// TIA Portal V15.1 export
// export: Created 2024-06-21T08:41:03.3487684Z, ExportSetting WithDefaults, DisplayName Totally Integrated Automation Portal, DisplayVersion V15.1 Update 5, DisplayName TIA Portal Openness, DisplayVersion V15.1 Update 5, DisplayName SINAMICS Startdrive Advanced, DisplayVersion V15.1, DisplayName G130, G150, S120, S150, SINAMICS MV, S210, DisplayVersion V15.1, DisplayName G110M, G120, G120C, G120D, G120P, DisplayVersion V15.1, DisplayName STEP 7 Professional, DisplayVersion V15.1 Update 5, DisplayName STEP 7 Safety, DisplayVersion V15.1, DisplayName WinCC Professional, DisplayVersion V15.1 Update 5, DisplayName SIMATIC Visualization Architect, DisplayVersion V15.1
FUNCTION_BLOCK "LProcMot1W-FCByp"   // FB1728, FBD
TITLE = LProcMotFCPidNoFbk
{ S7_Optimized_Access := 'FALSE' }
AUTHOR : VCC
FAMILY : ProcEq
NAME : FCPN
VERSION : 0.0
// ===============================================================================
// 
// This "Motor-1Way-1Speed-FreqCtrl with bypass module is used in applications 
// when 
// a motor 
// 1 way - 1 speed equipped with Danfoss equipment (FC) on
// Profibus or Profinet steering is needed.
// The module contains: 
// " 1selection 5 set point with 5 resonance 
// "1 mode from HMI
// "1 motor protection.
// "1 safety switch.
// "1 feedback motor running (option): Pressure-switch, Rotation guard,........
// "1 Proces Danfoss equipment with Profibus/Profinet.
// "1 bypass contactor.
// "1 bypass key-switch.
// ===============================================================================
// stored: AutoNumber false, IsIECCheckEnabled false, SetENOAutomatically False, UDAEnableTagReadback false
   VAR_INPUT
      I_ExtSP1_Value { ExternalAccessible := 'False'; ExternalVisible := 'False'; ExternalWritable := 'False'} : Real;   // External Set-point 1
      I_SPReq : Int;   // Index Set-point Request
      I_ExtSP1 { ExternalAccessible := 'False'; ExternalVisible := 'False'; ExternalWritable := 'False'} : Bool;   // External Set-point 1 Request
      I_EnableFCReset { ExternalAccessible := 'False'; ExternalVisible := 'False'; ExternalWritable := 'False'} : Bool;   // Enable Frequency reset with Fielbus
      I_EnableCheckSpeedOK { ExternalAccessible := 'False'; ExternalVisible := 'False'; ExternalWritable := 'False'} : Bool;   // Enable check speed is OK
      I_TimeCheckSpeedOK { ExternalAccessible := 'False'; ExternalVisible := 'False'; ExternalWritable := 'False'} : DInt := DINT#10000;   // Delay time to check if speed is OK
      I_RunFbkAlarmTime { ExternalAccessible := 'False'; ExternalVisible := 'False'; ExternalWritable := 'False'} : DInt;   // Time for alarm Feedback Motor running
      I_EnableAlarm { ExternalAccessible := 'False'; ExternalVisible := 'False'; ExternalWritable := 'False'} : Bool;   // Enable alarm
      I_AutoReq { ExternalAccessible := 'False'; ExternalVisible := 'False'; ExternalWritable := 'False'} : Bool;   // Auto Request from equation or Sequence
      I_InterlockOk { ExternalAccessible := 'False'; ExternalVisible := 'False'; ExternalWritable := 'False'} : Bool;   // Interlock Ok
      I_MotorProtection { ExternalAccessible := 'False'; ExternalVisible := 'False'; ExternalWritable := 'False'} : Bool;   // Motor protection Ok
      I_BypassKey { ExternalAccessible := 'False'; ExternalVisible := 'False'; ExternalWritable := 'False'} : Bool;   // Bypass Key-switch
      I_SafetySwitch { ExternalAccessible := 'False'; ExternalVisible := 'False'; ExternalWritable := 'False'} : Bool;   // Safety Switch Ok
      I_RunFeedBack { ExternalAccessible := 'False'; ExternalVisible := 'False'; ExternalWritable := 'False'} : Bool;   // Feedback motor running (Pressure-switch, Rotation Guard,...)
      I_PBSetPBResetAllAutoSel { ExternalAccessible := 'False'; ExternalVisible := 'False'; ExternalWritable := 'False'} : Struct   // Set PB activated - Reset PB activated - All HMI Auto selected
         HMI1SetPB { ExternalAccessible := 'False'; ExternalVisible := 'False'; ExternalWritable := 'False'} : Bool;   // Set PB activated on HMI1
         HMI1ResetPB { ExternalAccessible := 'False'; ExternalVisible := 'False'; ExternalWritable := 'False'} : Bool;   // Reset PB activated on HMI1
         HMI1AllHMIAutoSel { ExternalAccessible := 'False'; ExternalVisible := 'False'; ExternalWritable := 'False'} : Bool;   // All HMI Auto selected on HMI1
         HMI2SetPB { ExternalAccessible := 'False'; ExternalVisible := 'False'; ExternalWritable := 'False'} : Bool;   // Set PB activated on HMI2
         HMI2ResetPB { ExternalAccessible := 'False'; ExternalVisible := 'False'; ExternalWritable := 'False'} : Bool;   // Reset PB activated on HMI2
         HMI2AllHMIAutoSel { ExternalAccessible := 'False'; ExternalVisible := 'False'; ExternalWritable := 'False'} : Bool;   // All HMI Auto selected on HMI2
         HMI3SetPB { ExternalAccessible := 'False'; ExternalVisible := 'False'; ExternalWritable := 'False'} : Bool;   // Set PB activated on HMI3
         HMI3ResetPB { ExternalAccessible := 'False'; ExternalVisible := 'False'; ExternalWritable := 'False'} : Bool;   // Reset PB activated on HMI3
         HMI3AllHMIAutoSel { ExternalAccessible := 'False'; ExternalVisible := 'False'; ExternalWritable := 'False'} : Bool;   // All HMI Auto selected on HMI3
         HMI4SetPB { ExternalAccessible := 'False'; ExternalVisible := 'False'; ExternalWritable := 'False'} : Bool;   // Set PB activated on HMI4
         HMI4ResetPB { ExternalAccessible := 'False'; ExternalVisible := 'False'; ExternalWritable := 'False'} : Bool;   // Reset PB activated on HMI4
         HMI4AllHMIAutoSel { ExternalAccessible := 'False'; ExternalVisible := 'False'; ExternalWritable := 'False'} : Bool;   // All HMI Auto selected on HMI4
         HMI5SetPB { ExternalAccessible := 'False'; ExternalVisible := 'False'; ExternalWritable := 'False'} : Bool;   // Set PB activated on HMI5
         HMI5ResetPB { ExternalAccessible := 'False'; ExternalVisible := 'False'; ExternalWritable := 'False'} : Bool;   // Reset PB activated on HMI5
         HMI5AllHMIAutoSel { ExternalAccessible := 'False'; ExternalVisible := 'False'; ExternalWritable := 'False'} : Bool;   // All HMI Auto selected on HMI5
         StartPBSel { ExternalAccessible := 'False'; ExternalVisible := 'False'; ExternalWritable := 'False'} : Bool;   // Start is activated
         AlarmResetPBSel { ExternalAccessible := 'False'; ExternalVisible := 'False'; ExternalWritable := 'False'} : Bool;   // Alarm reset is activated
      END_STRUCT;
      I_UpperLevelAlarmA { ExternalAccessible := 'False'; ExternalVisible := 'False'; ExternalWritable := 'False'} : Bool;   // Upper level alarm A
      I_UpperLevelAlarmB { ExternalAccessible := 'False'; ExternalVisible := 'False'; ExternalWritable := 'False'} : Bool;   // Upper level alarm B
      I_HWSubInput { ExternalAccessible := 'False'; ExternalVisible := 'False'; ExternalWritable := 'False'} : HW_SUBMODULE;   // I/O connection hardware
      I_HWSubOutput { ExternalAccessible := 'False'; ExternalVisible := 'False'; ExternalWritable := 'False'} : HW_SUBMODULE;   // I/O connection hardware
      C_EnableSetResetHMI { ExternalAccessible := 'False'; ExternalVisible := 'False'; ExternalWritable := 'False'} : Bool;   // Enable Set-Reset functions from HMI
      C_SelfHolding { ExternalAccessible := 'False'; ExternalVisible := 'False'; ExternalWritable := 'False'} : Bool := TRUE;   // Enable SelfHolding Command
      C_RunFeedBackUsed { ExternalAccessible := 'False'; ExternalVisible := 'False'; ExternalWritable := 'False'} : Bool;   // Feedback motor running is used
      C_SafetySwNc { ExternalAccessible := 'False'; ExternalVisible := 'False'; ExternalWritable := 'False'} : Bool;   // Safety switch Normally closed
      C_MotorProtectionNc { ExternalAccessible := 'False'; ExternalVisible := 'False'; ExternalWritable := 'False'} : Bool;   // Motor protection Normally closed
      C_BypassSw_HW { ExternalAccessible := 'False'; ExternalVisible := 'False'; ExternalWritable := 'False'} : Bool := TRUE;   // Bypass-switch Hardware (=true) otherwise Software
      C_BypassSwOffFault { ExternalAccessible := 'False'; ExternalVisible := 'False'; ExternalWritable := 'False'} : Bool := TRUE;   // Bypass Switch active when input = False
      C_ManualForced { ExternalAccessible := 'False'; ExternalVisible := 'False'; ExternalWritable := 'False'} : Bool;   // Manual Forced is used (=true)
   END_VAR
   VAR_OUTPUT
      O_SP : Real;   // Setpoint used in controller
      O_Contactor { ExternalAccessible := 'False'; ExternalVisible := 'False'; ExternalWritable := 'False'} : Bool;   // Contactor of motor loop
      O_MotorRunning { ExternalAccessible := 'False'; ExternalVisible := 'False'; ExternalWritable := 'False'} : Bool;   // Motor is running
      O_AlarmABCondition { ExternalAccessible := 'False'; ExternalVisible := 'False'; ExternalWritable := 'False'} : Bool;   // Alarms resetable
      O_AlarmA { ExternalAccessible := 'False'; ExternalVisible := 'False'; ExternalWritable := 'False'} : Bool;   // Alarm A
      O_AlarmB { ExternalAccessible := 'False'; ExternalVisible := 'False'; ExternalWritable := 'False'} : Bool;   // Alarm B
      O_AlarmC { ExternalAccessible := 'False'; ExternalVisible := 'False'; ExternalWritable := 'False'} : Bool;   // Alarm C
      O_AlarmD { ExternalAccessible := 'False'; ExternalVisible := 'False'; ExternalWritable := 'False'} : Bool;   // Alarm D
      H_IAnim { ExternalAccessible := 'False'; ExternalVisible := 'False'; ExternalWritable := 'False'} : Word;   // HMI Animation color of the icon
      H_AlarmWord { ExternalAccessible := 'False'; ExternalVisible := 'False'; ExternalWritable := 'False'} : DWord;   // Alarm Word
   END_VAR
   VAR_IN_OUT
      FCDP : "LProcDanfoss";   // DB of submodule for the Frequency controller
   END_VAR
   VAR DB_SPECIFIC
      AA_MotorProtection { ExternalAccessible := 'False'; ExternalVisible := 'False'; ExternalWritable := 'False'} : Bool;   // Motor Protection alarm
      AA_SafetySwitch { ExternalAccessible := 'False'; ExternalVisible := 'False'; ExternalWritable := 'False'} : Bool;   // Safety Switch alarm
      AA_FreqController { ExternalAccessible := 'False'; ExternalVisible := 'False'; ExternalWritable := 'False'} : Bool;   // Frequency controller alarm A
      AB_RunFeedback { ExternalAccessible := 'False'; ExternalVisible := 'False'; ExternalWritable := 'False'} : Bool;   // Motor Running Feedback Alarm
      AB_OvTimeAutoSel { ExternalAccessible := 'False'; ExternalVisible := 'False'; ExternalWritable := 'False'} : Bool;   // Overtime Auto selected
      AC_FreqController { ExternalAccessible := 'False'; ExternalVisible := 'False'; ExternalWritable := 'False'} : Bool;   // Frequency controller alarm C
      AD_InterlockAlarm { ExternalAccessible := 'False'; ExternalVisible := 'False'; ExternalWritable := 'False'} : Bool;   // Interlock Alarm
      AD_BypassSwitch { ExternalAccessible := 'False'; ExternalVisible := 'False'; ExternalWritable := 'False'} : Bool;   // Bypass-Switch Alarm
      AD_BypassSoftKey { ExternalAccessible := 'False'; ExternalVisible := 'False'; ExternalWritable := 'False'} : Bool;   // Bypass-Key HMI Alarm
      H_HMIModeCmd : Word;   // Mode commands from HMI
      H_ActiveHMI : Int;   // Active HMI
      H_NameActiveHMI : String[25];   // Name of the Active HMI
      H_In : Struct   // HMI
         Normalbandwidthmode : Bool := TRUE;   // Each resonance frequency his own bandwidth
         SPResonance1 : Real;   // Set-point 1 Resonance frequency
         SPResonance2 : Real;   // Set-point 2 Resonance frequency
         SPResonance3 : Real;   // Set-point 3 Resonance frequency
         SPResonance4 : Real;   // Set-point 4 Resonance frequency
         SPBandwidth1 : Real;   // Set-point 1 Bandwidth (for resonance frequency)
         SPBandwidth2 : Real;   // Set-point 2 Bandwidth (for resonance frequency)
         SPBandwidth3 : Real;   // Set-point 3 Bandwidth (for resonance frequency)
         SPBandwidth4 : Real;   // Set-point 4 Bandwidth (for resonance frequency)
      END_STRUCT;
      H_Out : Struct   // HMI
         MotorProtectIAnim : Word;   // HMI Animation color of object
         SafetySwitchIAnim : Word;   // HMI Animation color of object
         FCIAnim : Word;   // HMI Animation color of object
         ContactorIAnim : Word;   // HMI Animation color of object
         BypassSwitchIAnim : Word;   // HMI Animation color of object
         RunFbkIAnim : Word;   // HMI Animation color of object
         Anim : Word;   // HMI Animation word
         Anim2 : Word;   // HMI Animation word
         Anim3 : Bool;   // HMI Animation bool
         DBnr : Int;   // HMI Animation DB number
      END_STRUCT;
      H_InOut : Struct   // HMI
         SetpntAllowed : Bool := TRUE;   // Setpoint is OK and allowed
         Manual_Value : Real;   // Position Setpoint in Manual
         SP1 : Real;   // Set-point 1
         SP2 : Real;   // Set-point 2
         SP3 : Real;   // Set-point 3
         SP4 : Real;   // Set-point 4
         SP5 : Real;   // Set-point 5
      END_STRUCT;
      AutoMode { ExternalAccessible := 'False'; ExternalVisible := 'False'; ExternalWritable := 'False'} : Bool;   // Auto mode
      ManualMode { ExternalAccessible := 'False'; ExternalVisible := 'False'; ExternalWritable := 'False'} : Bool;   // Manual mode
      AutoModeSel { ExternalAccessible := 'False'; ExternalVisible := 'False'; ExternalWritable := 'False'} : Bool;   // Auto Mode Selection from HMI
      ManualModeSel { ExternalAccessible := 'False'; ExternalVisible := 'False'; ExternalWritable := 'False'} : Bool;   // Manual Mode Selection from HMI
      HMISetCmd { ExternalAccessible := 'False'; ExternalVisible := 'False'; ExternalWritable := 'False'} : Bool;   // Set Command on HMI
      HMIResetCmd { ExternalAccessible := 'False'; ExternalVisible := 'False'; ExternalWritable := 'False'} : Bool;   // Reset Command on HMI
      H_FncSelInHMI { ExternalAccessible := 'False'; ExternalVisible := 'False'; ExternalWritable := 'False'} : Bool;   // Manual selection from HMI
      ForcedMan { ExternalAccessible := 'False'; ExternalVisible := 'False'; ExternalWritable := 'False'} : Bool;   // Forced manual active
      OvTimeAutoSel { ExternalAccessible := 'False'; ExternalVisible := 'False'; ExternalWritable := 'False'} : Bool;   // Overtime Auto selected
      OvTimeAutoSelCond { ExternalAccessible := 'False'; ExternalVisible := 'False'; ExternalWritable := 'False'} : Bool;   // Overtime Auto selected condition
      MotorProtectionABCond { ExternalAccessible := 'False'; ExternalVisible := 'False'; ExternalWritable := 'False'} : Bool;   // Motor protection alarm can be reset
      MotorProtectionDisable { ExternalAccessible := 'False'; ExternalVisible := 'False'; ExternalWritable := 'False'} : Bool;   // Motor protection alarm is disabled from HMI
      SafetySwitchABCond { ExternalAccessible := 'False'; ExternalVisible := 'False'; ExternalWritable := 'False'} : Bool;   // Safety Switch alarm can be reset
      SafetySwitchDisable { ExternalAccessible := 'False'; ExternalVisible := 'False'; ExternalWritable := 'False'} : Bool;   // Safety Switch alarm is disabled from HMI
      StartCmdFC { ExternalAccessible := 'False'; ExternalVisible := 'False'; ExternalWritable := 'False'} : Bool;   // Start Command Frequency controller signal
      MRV_FC { ExternalAccessible := 'False'; ExternalVisible := 'False'; ExternalWritable := 'False'} : Int;   // Frequency controller MRV (main reference value)
      FCActive { ExternalAccessible := 'False'; ExternalVisible := 'False'; ExternalWritable := 'False'} : Bool;   // Frequency controller - Profibus active
      FCAlarmDisable { ExternalAccessible := 'False'; ExternalVisible := 'False'; ExternalWritable := 'False'} : Bool;   // Frequency controller alarms are disable from HMI
      FCABCond { ExternalAccessible := 'False'; ExternalVisible := 'False'; ExternalWritable := 'False'} : Bool;   // Frequency controller alarm can be reset
      BypassSwitchDisable { ExternalAccessible := 'False'; ExternalVisible := 'False'; ExternalWritable := 'False'} : Bool;   // Bypass-switch alarm is disabled from HMI
      BypassForced { ExternalAccessible := 'False'; ExternalVisible := 'False'; ExternalWritable := 'False'} : Bool;   // Bypass Forced by Key-switch
      RunFbkEnAlarm { ExternalAccessible := 'False'; ExternalVisible := 'False'; ExternalWritable := 'False'} : Bool;   // Motor Running Feedback Enable Alarm
      RunFbkDisable { ExternalAccessible := 'False'; ExternalVisible := 'False'; ExternalWritable := 'False'} : Bool;   // Motor Running Feedback Alarm is disabled from HMI
      RunFeedBackABCond { ExternalAccessible := 'False'; ExternalVisible := 'False'; ExternalWritable := 'False'} : Bool;   // Motor Running Feedback Alarm can be reset
      CmdRequest { ExternalAccessible := 'False'; ExternalVisible := 'False'; ExternalWritable := 'False'} : Bool;   // Command request to activate the component
      SetPBMan { ExternalAccessible := 'False'; ExternalVisible := 'False'; ExternalWritable := 'False'} : Bool;   // Set pushbutton is activated in manual
      ResetPBMan { ExternalAccessible := 'False'; ExternalVisible := 'False'; ExternalWritable := 'False'} : Bool;   // Reset pushbutton is activated in manual
      AllHMIAutoSel { ExternalAccessible := 'False'; ExternalVisible := 'False'; ExternalWritable := 'False'} : Bool;   // All HMI Auto selected
      Active { ExternalAccessible := 'False'; ExternalVisible := 'False'; ExternalWritable := 'False'} : Bool;   // Motor Loop is active
      Contactor { ExternalAccessible := 'False'; ExternalVisible := 'False'; ExternalWritable := 'False'} : Bool;   // Contactor
      SPSel { ExternalAccessible := 'False'; ExternalVisible := 'False'; ExternalWritable := 'False'} : Real;   // Set-point selected
      SPReal { ExternalAccessible := 'False'; ExternalVisible := 'False'; ExternalWritable := 'False'} : Real;   // Manual or Automatic Set-point selected Real
      SPDINT { ExternalAccessible := 'False'; ExternalVisible := 'False'; ExternalWritable := 'False'} : DInt;   // Set-point selected DInteger
      AlarmA { ExternalAccessible := 'False'; ExternalVisible := 'False'; ExternalWritable := 'False'} : Bool;   // Summation Alarm A
      AlarmB { ExternalAccessible := 'False'; ExternalVisible := 'False'; ExternalWritable := 'False'} : Bool;   // Summation Alarm B
      AlarmC { ExternalAccessible := 'False'; ExternalVisible := 'False'; ExternalWritable := 'False'} : Bool;   // Summation Alarm C
      AlarmD { ExternalAccessible := 'False'; ExternalVisible := 'False'; ExternalWritable := 'False'} : Bool;   // Summation Alarm D
      DBnr { ExternalAccessible := 'False'; ExternalVisible := 'False'; ExternalWritable := 'False'} : Int;   // HMI DB number
   END_VAR
   VAR
      RunFbkTimer { ExternalAccessible := 'False'; ExternalVisible := 'False'; ExternalWritable := 'False'; S7_SetPoint := 'True'} : "LTimer";   // Timer Run Feedback Alarm
      RunFeedback { ExternalAccessible := 'False'; ExternalVisible := 'False'; ExternalWritable := 'False'; S7_SetPoint := 'True'} : "LProc1AlarmMultiIn";   // Run Feedback Alarm
      MotorProtection { ExternalAccessible := 'False'; ExternalVisible := 'False'; ExternalWritable := 'False'; S7_SetPoint := 'True'} : "LProc1AlarmMultiIn";   // Motor protection alarm
      SafetySwitch { ExternalAccessible := 'False'; ExternalVisible := 'False'; ExternalWritable := 'False'; S7_SetPoint := 'True'} : "LProc1AlarmMultiIn";   // Safety Switch alarm
      BypassSwitch { ExternalAccessible := 'False'; ExternalVisible := 'False'; ExternalWritable := 'False'; S7_SetPoint := 'True'} : "LProc1AlarmMultiIn";   // Bypass alarm
      Modes { ExternalAccessible := 'False'; ExternalVisible := 'False'; ExternalWritable := 'False'; S7_SetPoint := 'True'} : "LProcObjectMode";   // Modes Handling
      SelSp { ExternalAccessible := 'False'; ExternalVisible := 'False'; ExternalWritable := 'False'; S7_SetPoint := 'True'} : "LProcSel5SPResFreq";
   END_VAR
   VAR DB_SPECIFIC
      CheckActiveHMI { ExternalAccessible := 'False'; ExternalVisible := 'False'; ExternalWritable := 'False'; S7_SetPoint := 'True'} : TP_TIME;   // Timer
      CheckActiveHMI_1 { ExternalAccessible := 'False'; ExternalVisible := 'False'; ExternalWritable := 'False'; S7_SetPoint := 'True'} : TP_TIME;   // Timer
      CheckActiveHMI_2 { ExternalAccessible := 'False'; ExternalVisible := 'False'; ExternalWritable := 'False'; S7_SetPoint := 'True'} : TON_TIME;   // Timer
      CheckActiveHMI_3 { ExternalAccessible := 'False'; ExternalVisible := 'False'; ExternalWritable := 'False'; S7_SetPoint := 'True'} : TON_TIME;   // Timer
   END_VAR
   VAR_TEMP
      __PlcmigTempFillBits_0B0 : Array[0..23] of Bool;
   END_VAR
BEGIN

NETWORK
TITLE = **** 1 - Inputs **** DB number
// DB number
      L     DINO;
      T     #DBnr;

REGION Network 2: **** 1 - Inputs **** Extract the command bits from HMI
   // Extract the command bits from HMI
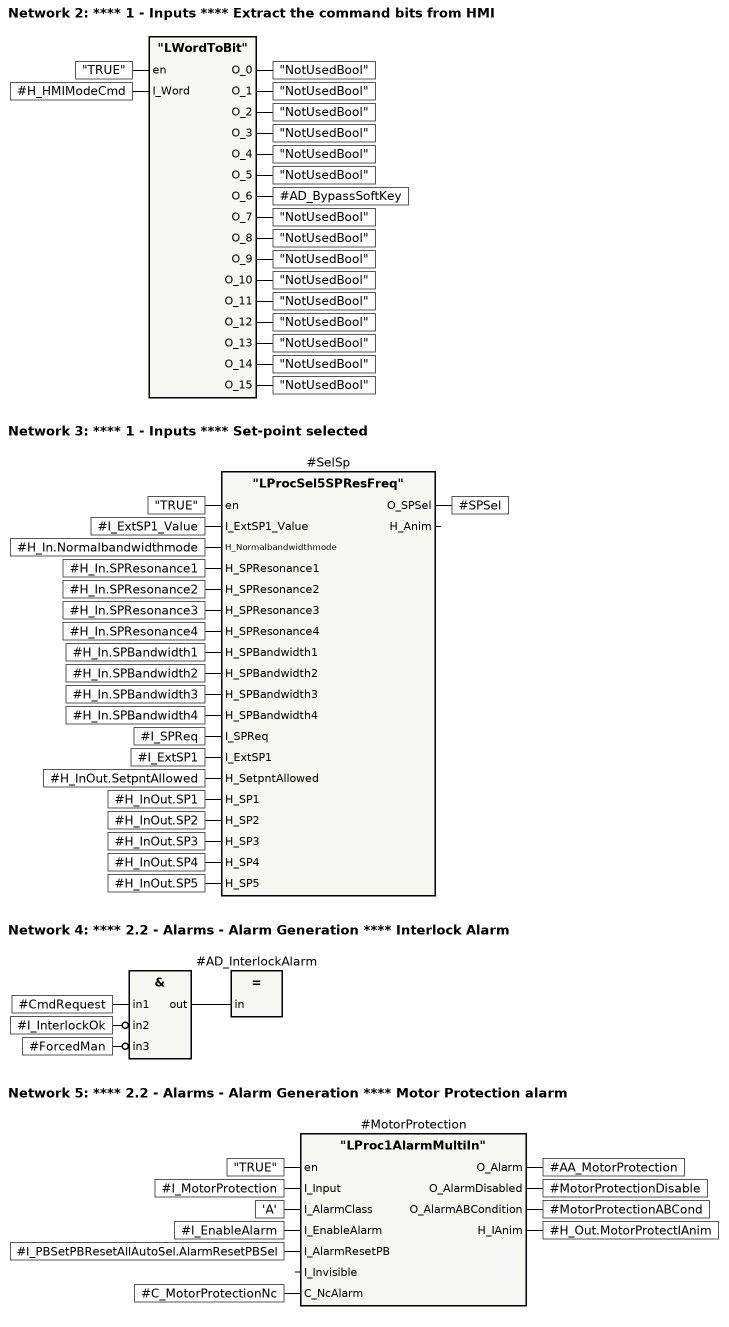
   IF "TRUE" THEN
       "LWordToBit"(I_Word := #H_HMIModeCmd,
                    O_0 => "NotUsedBool",
                    O_1 => "NotUsedBool",
                    O_2 => "NotUsedBool",
                    O_3 => "NotUsedBool",
                    O_4 => "NotUsedBool",
                    O_5 => "NotUsedBool",
                    O_6 => #AD_BypassSoftKey,
                    O_7 => "NotUsedBool",
                    O_8 => "NotUsedBool",
                    O_9 => "NotUsedBool",
                    O_10 => "NotUsedBool",
                    O_11 => "NotUsedBool",
                    O_12 => "NotUsedBool",
                    O_13 => "NotUsedBool",
                    O_14 => "NotUsedBool",
                    O_15 => "NotUsedBool");
   END_IF;
END_REGION

REGION Network 3: **** 1 - Inputs **** Set-point selected
   // Set-point selected
   IF "TRUE" THEN
       #SelSp(I_ExtSP1_Value := #I_ExtSP1_Value,   // "LProcSel5SPResFreq"
              H_Normalbandwidthmode := #H_In.Normalbandwidthmode,
              H_SPResonance1 := #H_In.SPResonance1,
              H_SPResonance2 := #H_In.SPResonance2,
              H_SPResonance3 := #H_In.SPResonance3,
              H_SPResonance4 := #H_In.SPResonance4,
              H_SPBandwidth1 := #H_In.SPBandwidth1,
              H_SPBandwidth2 := #H_In.SPBandwidth2,
              H_SPBandwidth3 := #H_In.SPBandwidth3,
              H_SPBandwidth4 := #H_In.SPBandwidth4,
              I_SPReq := #I_SPReq,
              I_ExtSP1 := #I_ExtSP1,
              H_SetpntAllowed := #H_InOut.SetpntAllowed,
              H_SP1 := #H_InOut.SP1,
              H_SP2 := #H_InOut.SP2,
              H_SP3 := #H_InOut.SP3,
              H_SP4 := #H_InOut.SP4,
              H_SP5 := #H_InOut.SP5,
              O_SPSel => #SPSel);
   END_IF;
END_REGION

REGION Network 4: **** 2.2 - Alarms - Alarm Generation **** Interlock Alarm
   // Interlock Alarm
   #AD_InterlockAlarm := #CmdRequest AND NOT #I_InterlockOk AND NOT #ForcedMan;
END_REGION

REGION Network 5: **** 2.2 - Alarms - Alarm Generation **** Motor Protection alarm
   // Motor Protection alarm
   IF "TRUE" THEN
       #MotorProtection(I_Input := #I_MotorProtection,   // "LProc1AlarmMultiIn"
                        I_AlarmClass := 'A',
                        I_EnableAlarm := #I_EnableAlarm,
                        I_AlarmResetPB := #I_PBSetPBResetAllAutoSel.AlarmResetPBSel,
                        C_NcAlarm := #C_MotorProtectionNc,
                        O_Alarm => #AA_MotorProtection,
                        O_AlarmDisabled => #MotorProtectionDisable,
                        O_AlarmABCondition => #MotorProtectionABCond,
                        H_IAnim => #H_Out.MotorProtectIAnim);
   END_IF;
END_REGION

REGION Network 6: **** 2.2 - Alarms - Alarm Generation **** Safety Switch alarm
   // Safety Switch alarm
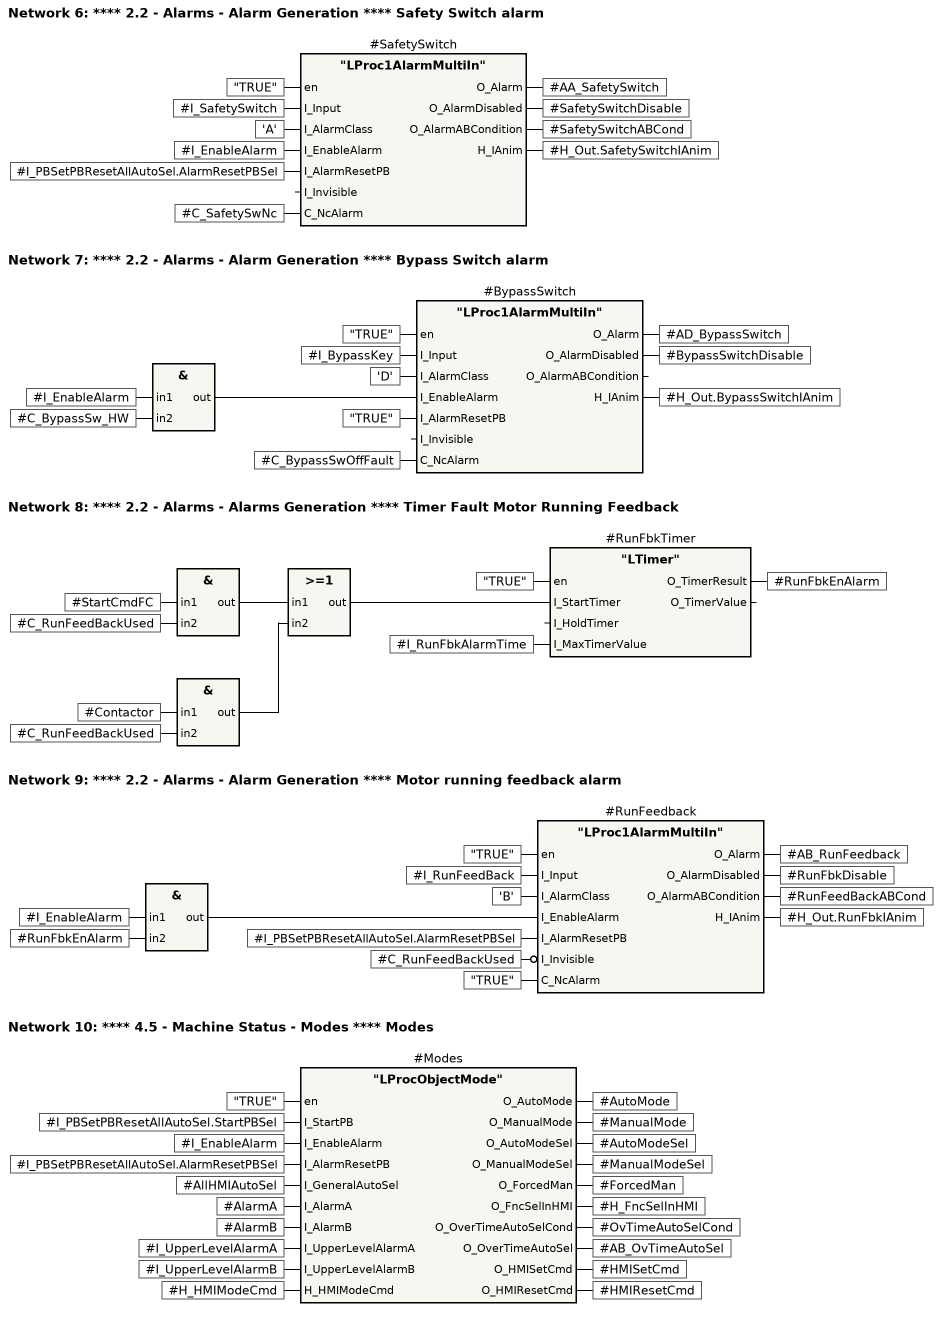
   IF "TRUE" THEN
       #SafetySwitch(I_Input := #I_SafetySwitch,   // "LProc1AlarmMultiIn"
                     I_AlarmClass := 'A',
                     I_EnableAlarm := #I_EnableAlarm,
                     I_AlarmResetPB := #I_PBSetPBResetAllAutoSel.AlarmResetPBSel,
                     C_NcAlarm := #C_SafetySwNc,
                     O_Alarm => #AA_SafetySwitch,
                     O_AlarmDisabled => #SafetySwitchDisable,
                     O_AlarmABCondition => #SafetySwitchABCond,
                     H_IAnim => #H_Out.SafetySwitchIAnim);
   END_IF;
END_REGION

REGION Network 7: **** 2.2 - Alarms - Alarm Generation **** Bypass Switch alarm
   // Bypass Switch alarm
   IF "TRUE" THEN
       #BypassSwitch(I_Input := #I_BypassKey,   // "LProc1AlarmMultiIn"
                     I_AlarmClass := 'D',
                     I_EnableAlarm := #I_EnableAlarm AND #C_BypassSw_HW,
                     I_AlarmResetPB := "TRUE",
                     C_NcAlarm := #C_BypassSwOffFault,
                     O_Alarm => #AD_BypassSwitch,
                     O_AlarmDisabled => #BypassSwitchDisable,
                     H_IAnim => #H_Out.BypassSwitchIAnim);
   END_IF;
END_REGION

REGION Network 8: **** 2.2 - Alarms - Alarms Generation **** Timer Fault Motor Running Feedback
   // Timer Fault Motor Running Feedback
   IF "TRUE" THEN
       #RunFbkTimer(I_StartTimer := (#StartCmdFC AND #C_RunFeedBackUsed) OR (#Contactor AND #C_RunFeedBackUsed),   // "LTimer"
                    I_MaxTimerValue := #I_RunFbkAlarmTime,
                    O_TimerResult => #RunFbkEnAlarm);
   END_IF;
END_REGION

REGION Network 9: **** 2.2 - Alarms - Alarm Generation **** Motor running feedback alarm
   // Motor running feedback alarm
   IF "TRUE" THEN
       #RunFeedback(I_Input := #I_RunFeedBack,   // "LProc1AlarmMultiIn"
                    I_AlarmClass := 'B',
                    I_EnableAlarm := #I_EnableAlarm AND #RunFbkEnAlarm,
                    I_AlarmResetPB := #I_PBSetPBResetAllAutoSel.AlarmResetPBSel,
                    I_Invisible := NOT #C_RunFeedBackUsed,
                    C_NcAlarm := "TRUE",
                    O_Alarm => #AB_RunFeedback,
                    O_AlarmDisabled => #RunFbkDisable,
                    O_AlarmABCondition => #RunFeedBackABCond,
                    H_IAnim => #H_Out.RunFbkIAnim);
   END_IF;
END_REGION

REGION Network 10: **** 4.5 - Machine Status - Modes **** Modes
   // Modes
   IF "TRUE" THEN
       #Modes(I_StartPB := #I_PBSetPBResetAllAutoSel.StartPBSel,   // "LProcObjectMode"
              I_EnableAlarm := #I_EnableAlarm,
              I_AlarmResetPB := #I_PBSetPBResetAllAutoSel.AlarmResetPBSel,
              I_GeneralAutoSel := #AllHMIAutoSel,
              I_AlarmA := #AlarmA,
              I_AlarmB := #AlarmB,
              I_UpperLevelAlarmA := #I_UpperLevelAlarmA,
              I_UpperLevelAlarmB := #I_UpperLevelAlarmB,
              H_HMIModeCmd := #H_HMIModeCmd,
              O_AutoMode => #AutoMode,
              O_ManualMode => #ManualMode,
              O_AutoModeSel => #AutoModeSel,
              O_ManualModeSel => #ManualModeSel,
              O_ForcedMan => #ForcedMan,
              O_FncSelInHMI => #H_FncSelInHMI,
              O_OverTimeAutoSelCond => #OvTimeAutoSelCond,
              O_OverTimeAutoSel => #AB_OvTimeAutoSel,
              O_HMISetCmd => #HMISetCmd,
              O_HMIResetCmd => #HMIResetCmd);
   END_IF;
END_REGION

REGION Network 11: **** 4.6 - Machine status - Indications **** Active
   // Active
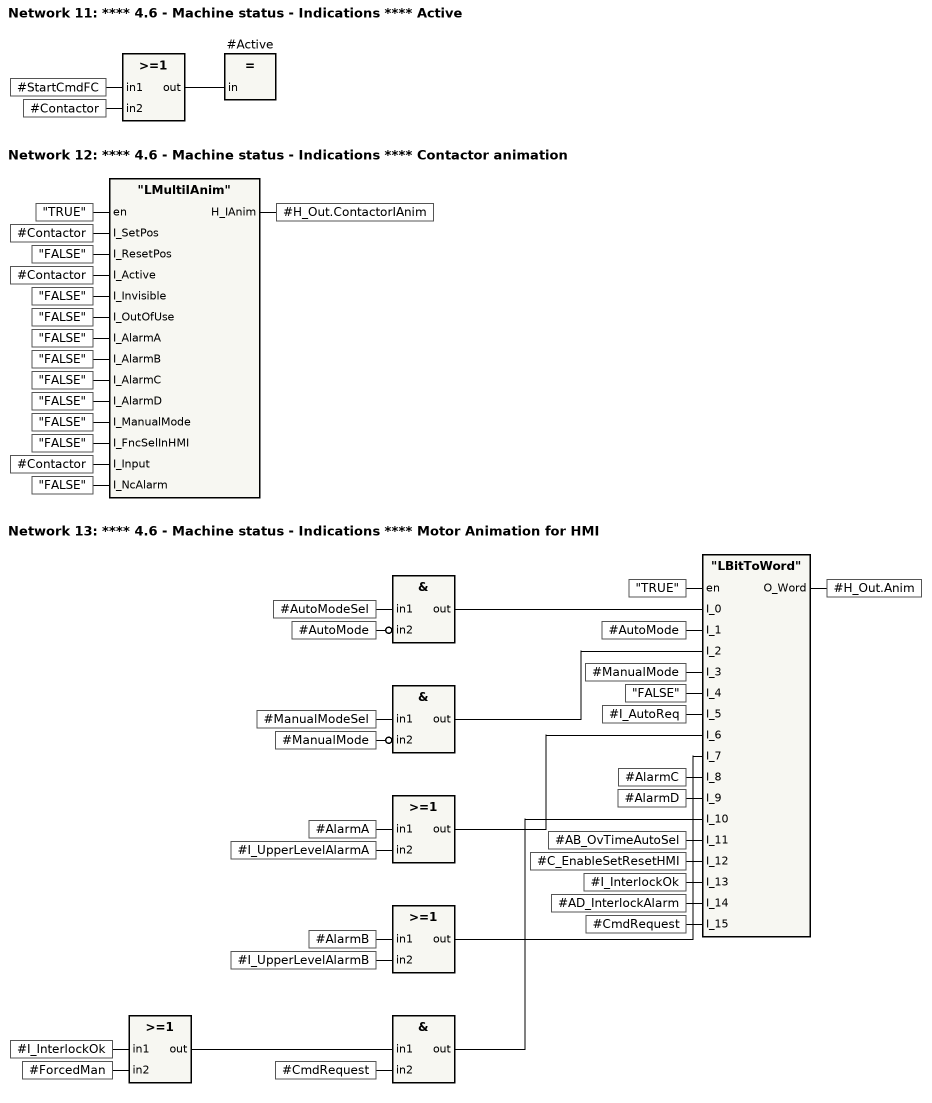
   #Active := #StartCmdFC OR #Contactor;
END_REGION

REGION Network 12: **** 4.6 - Machine status - Indications **** Contactor animation
   // Contactor animation
   IF "TRUE" THEN
       "LMultiIAnim"(I_SetPos := #Contactor,
                     I_ResetPos := "FALSE",
                     I_Active := #Contactor,
                     I_Invisible := "FALSE",
                     I_OutOfUse := "FALSE",
                     I_AlarmA := "FALSE",
                     I_AlarmB := "FALSE",
                     I_AlarmC := "FALSE",
                     I_AlarmD := "FALSE",
                     I_ManualMode := "FALSE",
                     I_FncSelInHMI := "FALSE",
                     I_Input := #Contactor,
                     I_NcAlarm := "FALSE",
                     H_IAnim => #H_Out.ContactorIAnim);
   END_IF;
END_REGION

REGION Network 13: **** 4.6 - Machine status - Indications **** Motor Animation for HMI
   // Motor Animation for HMI
   IF "TRUE" THEN
       "LBitToWord"(I_0 := #AutoModeSel AND NOT #AutoMode,
                    I_1 := #AutoMode,
                    I_2 := #ManualModeSel AND NOT #ManualMode,
                    I_3 := #ManualMode,
                    I_4 := "FALSE",
                    I_5 := #I_AutoReq,
                    I_6 := #AlarmA OR #I_UpperLevelAlarmA,
                    I_7 := #AlarmB OR #I_UpperLevelAlarmB,
                    I_8 := #AlarmC,
                    I_9 := #AlarmD,
                    I_10 := (#I_InterlockOk OR #ForcedMan) AND #CmdRequest,
                    I_11 := #AB_OvTimeAutoSel,
                    I_12 := #C_EnableSetResetHMI,
                    I_13 := #I_InterlockOk,
                    I_14 := #AD_InterlockAlarm,
                    I_15 := #CmdRequest,
                    O_Word => #H_Out.Anim);
   END_IF;
END_REGION

REGION Network 14: **** 4.6 - Machine status - Indications **** Motor Animation for HMI
   // Motor Animation for HMI
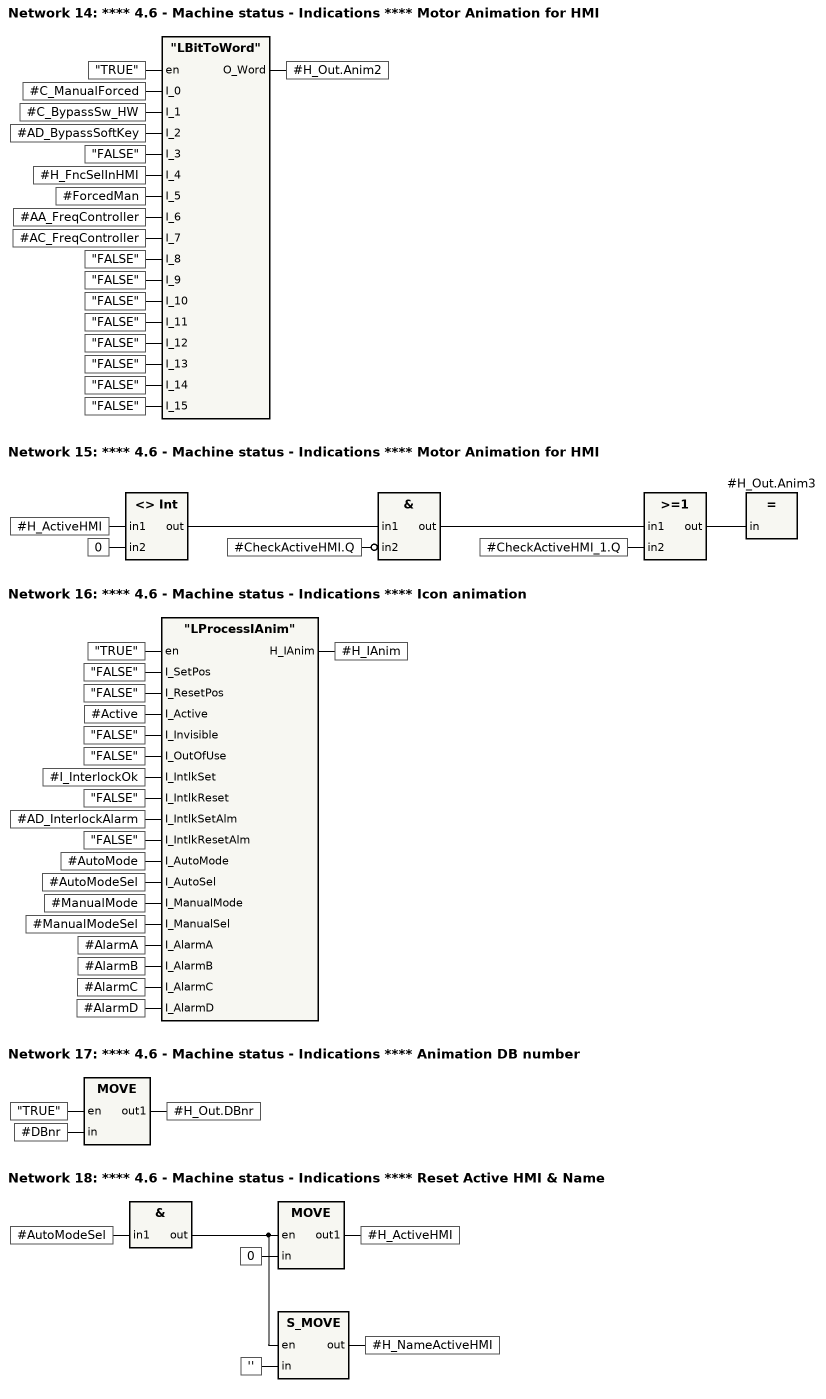
   IF "TRUE" THEN
       "LBitToWord"(I_0 := #C_ManualForced,
                    I_1 := #C_BypassSw_HW,
                    I_2 := #AD_BypassSoftKey,
                    I_3 := "FALSE",
                    I_4 := #H_FncSelInHMI,
                    I_5 := #ForcedMan,
                    I_6 := #AA_FreqController,
                    I_7 := #AC_FreqController,
                    I_8 := "FALSE",
                    I_9 := "FALSE",
                    I_10 := "FALSE",
                    I_11 := "FALSE",
                    I_12 := "FALSE",
                    I_13 := "FALSE",
                    I_14 := "FALSE",
                    I_15 := "FALSE",
                    O_Word => #H_Out.Anim2);
   END_IF;
END_REGION

REGION Network 15: **** 4.6 - Machine status - Indications **** Motor Animation for HMI
   // Motor Animation for HMI
   #H_Out.Anim3 := ((#H_ActiveHMI <> 0) AND NOT #CheckActiveHMI.Q) OR #CheckActiveHMI_1.Q;
END_REGION

REGION Network 16: **** 4.6 - Machine status - Indications **** Icon animation
   // Icon animation
   IF "TRUE" THEN
       "LProcessIAnim"(I_SetPos := "FALSE",
                       I_ResetPos := "FALSE",
                       I_Active := #Active,
                       I_Invisible := "FALSE",
                       I_OutOfUse := "FALSE",
                       I_IntlkSet := #I_InterlockOk,
                       I_IntlkReset := "FALSE",
                       I_IntlkSetAlm := #AD_InterlockAlarm,
                       I_IntlkResetAlm := "FALSE",
                       I_AutoMode := #AutoMode,
                       I_AutoSel := #AutoModeSel,
                       I_ManualMode := #ManualMode,
                       I_ManualSel := #ManualModeSel,
                       I_AlarmA := #AlarmA,
                       I_AlarmB := #AlarmB,
                       I_AlarmC := #AlarmC,
                       I_AlarmD := #AlarmD,
                       H_IAnim => #H_IAnim);
   END_IF;
END_REGION

REGION Network 17: **** 4.6 - Machine status - Indications **** Animation DB number
   // Animation DB number
   IF "TRUE" THEN #H_Out.DBnr := #DBnr; END_IF;
END_REGION

REGION Network 18: **** 4.6 - Machine status - Indications **** Reset Active HMI & Name
   // Reset Active HMI & Name
   IF #AutoModeSel THEN
       #H_ActiveHMI := 0;
       #H_NameActiveHMI := '';
   END_IF;
END_REGION

REGION Network 19: **** 5.2 - Equations - Flow **** Manual mode is active and the Set button is pressed
   // Manual mode is active and the Set button is pressed
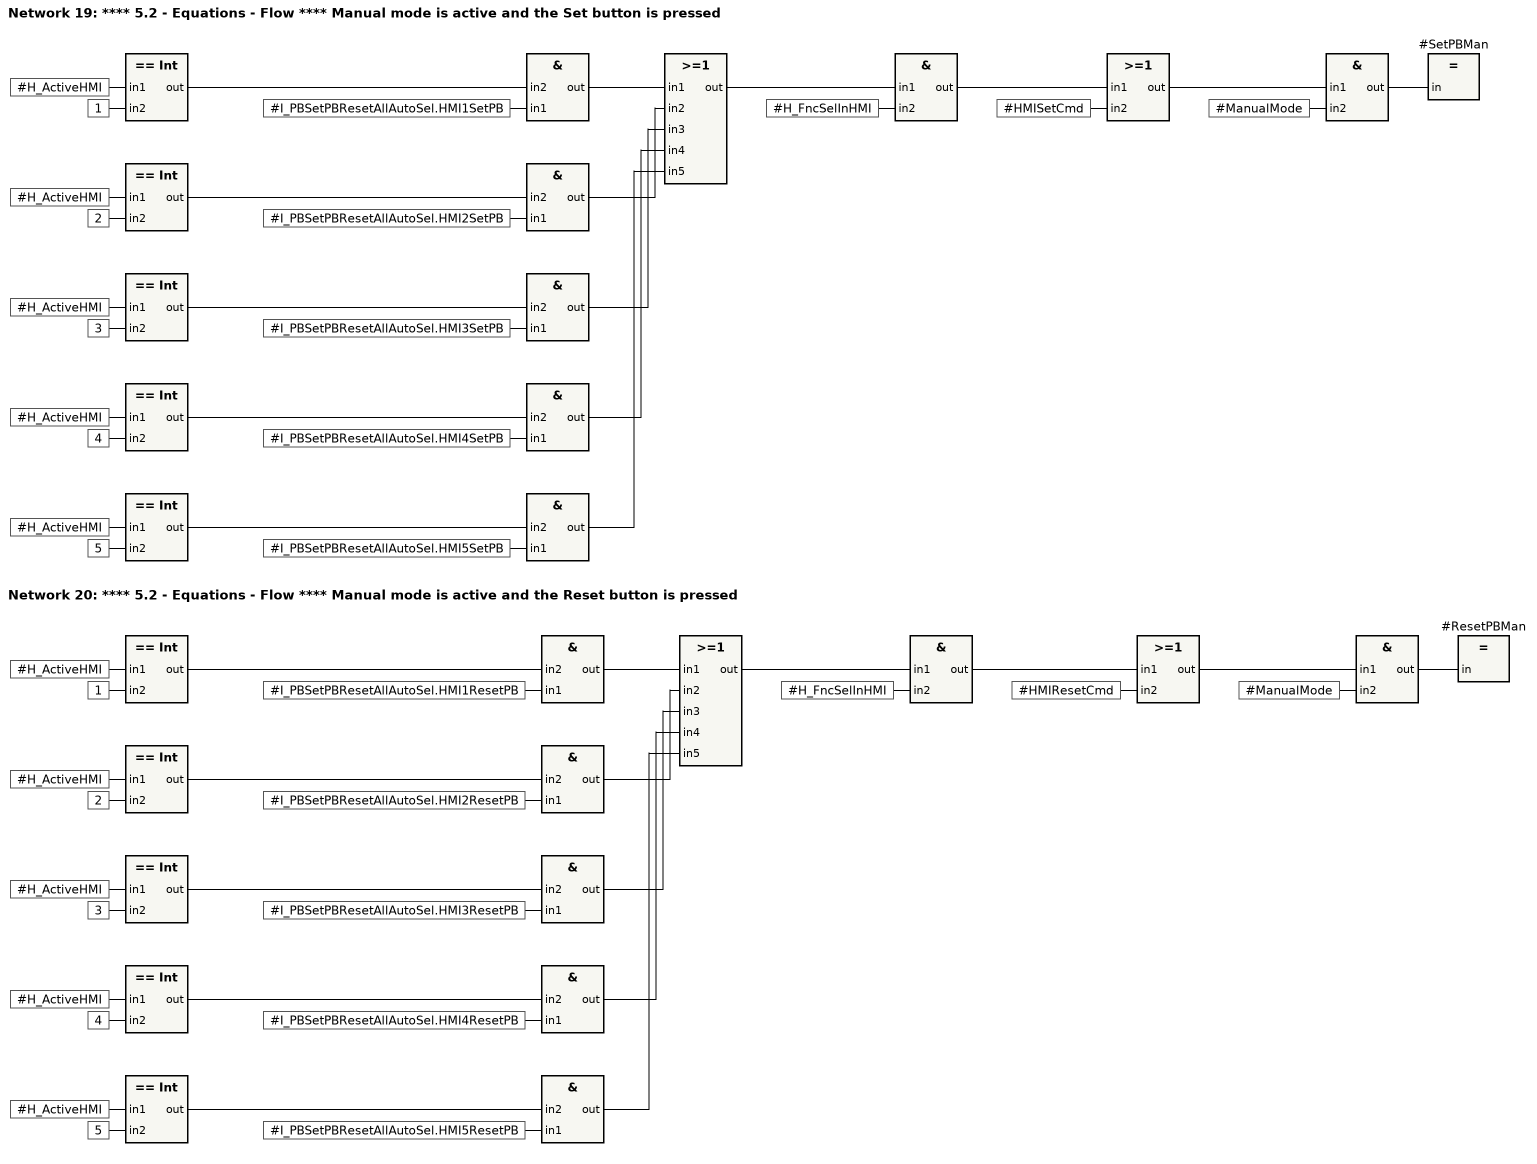
   #SetPBMan := (((((#H_ActiveHMI = 1) AND #I_PBSetPBResetAllAutoSel.HMI1SetPB) OR ((#H_ActiveHMI = 2) AND #I_PBSetPBResetAllAutoSel.HMI2SetPB) OR ((#H_ActiveHMI = 3) AND #I_PBSetPBResetAllAutoSel.HMI3SetPB) OR ((#H_ActiveHMI = 4) AND #I_PBSetPBResetAllAutoSel.HMI4SetPB) OR ((#H_ActiveHMI = 5) AND #I_PBSetPBResetAllAutoSel.HMI5SetPB)) AND #H_FncSelInHMI) OR #HMISetCmd) AND #ManualMode;
END_REGION

REGION Network 20: **** 5.2 - Equations - Flow **** Manual mode is active and the Reset button is pressed
   // Manual mode is active and the Reset button is pressed
   #ResetPBMan := (((((#H_ActiveHMI = 1) AND #I_PBSetPBResetAllAutoSel.HMI1ResetPB) OR ((#H_ActiveHMI = 2) AND #I_PBSetPBResetAllAutoSel.HMI2ResetPB) OR ((#H_ActiveHMI = 3) AND #I_PBSetPBResetAllAutoSel.HMI3ResetPB) OR ((#H_ActiveHMI = 4) AND #I_PBSetPBResetAllAutoSel.HMI4ResetPB) OR ((#H_ActiveHMI = 5) AND #I_PBSetPBResetAllAutoSel.HMI5ResetPB)) AND #H_FncSelInHMI) OR #HMIResetCmd) AND #ManualMode;
END_REGION

REGION Network 21: **** 5.2 - Equations - Flow **** All HMI Auto selected
   // All HMI Auto selected
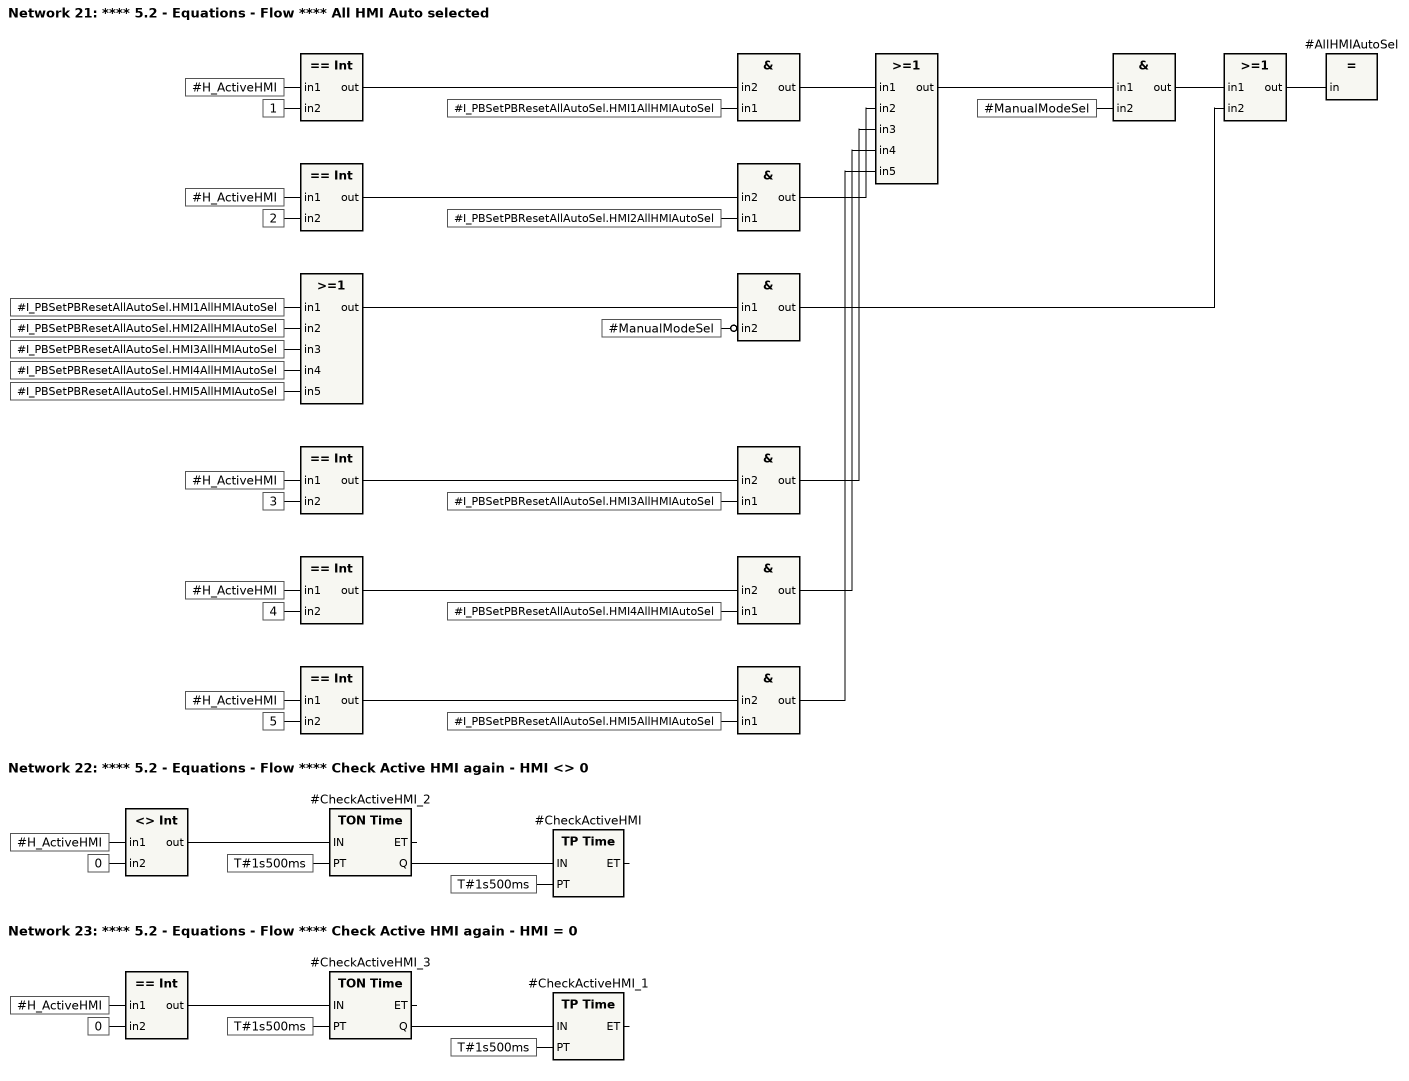
   #AllHMIAutoSel := ((((#H_ActiveHMI = 1) AND #I_PBSetPBResetAllAutoSel.HMI1AllHMIAutoSel) OR ((#H_ActiveHMI = 2) AND #I_PBSetPBResetAllAutoSel.HMI2AllHMIAutoSel) OR ((#H_ActiveHMI = 3) AND #I_PBSetPBResetAllAutoSel.HMI3AllHMIAutoSel) OR ((#H_ActiveHMI = 4) AND #I_PBSetPBResetAllAutoSel.HMI4AllHMIAutoSel) OR ((#H_ActiveHMI = 5) AND #I_PBSetPBResetAllAutoSel.HMI5AllHMIAutoSel)) AND #ManualModeSel) OR ((#I_PBSetPBResetAllAutoSel.HMI1AllHMIAutoSel OR #I_PBSetPBResetAllAutoSel.HMI2AllHMIAutoSel OR #I_PBSetPBResetAllAutoSel.HMI3AllHMIAutoSel OR #I_PBSetPBResetAllAutoSel.HMI4AllHMIAutoSel OR #I_PBSetPBResetAllAutoSel.HMI5AllHMIAutoSel) AND NOT #ManualModeSel);
END_REGION

REGION Network 22: **** 5.2 - Equations - Flow **** Check Active HMI again - HMI <> 0
   // Check Active HMI again
   #CheckActiveHMI_2(IN := #H_ActiveHMI <> 0, PT := T#1s500ms);   // TON
   #CheckActiveHMI(IN := #CheckActiveHMI_2.Q, PT := T#1s500ms);   // TP
END_REGION

REGION Network 23: **** 5.2 - Equations - Flow **** Check Active HMI again - HMI = 0
   // Check Active HMI again
   #CheckActiveHMI_3(IN := #H_ActiveHMI = 0, PT := T#1s500ms);   // TON
   #CheckActiveHMI_1(IN := #CheckActiveHMI_3.Q, PT := T#1s500ms);   // TP
END_REGION

REGION Network 24: **** 7.3 - Submodule - Machine **** Command Request
   // Command Request
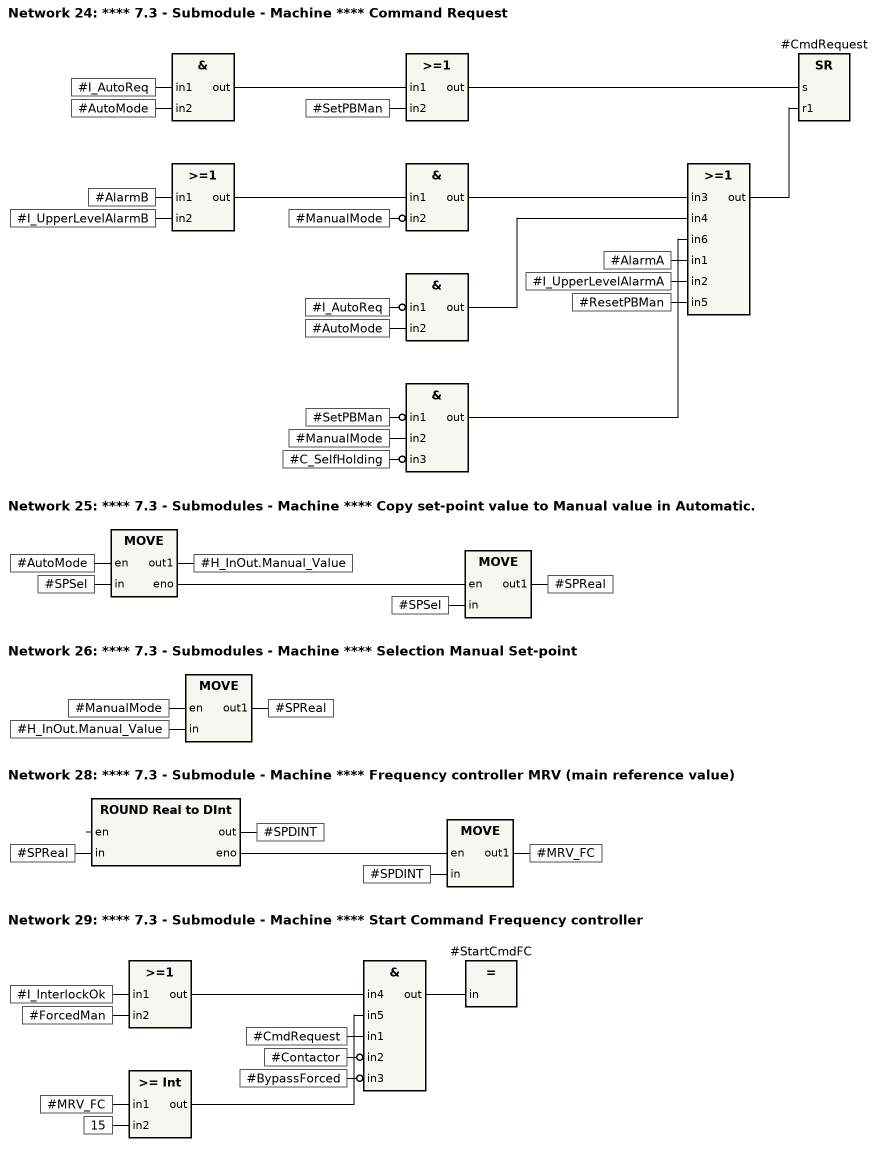
   IF (#I_AutoReq AND #AutoMode) OR #SetPBMan THEN
       #CmdRequest := TRUE;   // SR flip-flop
   END_IF;
   IF ((#AlarmB OR #I_UpperLevelAlarmB) AND NOT #ManualMode) OR (NOT #I_AutoReq AND #AutoMode) OR (NOT #SetPBMan AND #ManualMode AND NOT #C_SelfHolding) OR #AlarmA OR #I_UpperLevelAlarmA OR #ResetPBMan THEN
       #CmdRequest := FALSE;
   END_IF;
END_REGION

REGION Network 25: **** 7.3 - Submodules - Machine **** Copy set-point value to Manual value in Automatic.
   // Copy set-point value to Manual value in Automatic.
   // ENO of a box is taken as its EN; it also drops when the box reports an error
   IF #AutoMode THEN
       #H_InOut.Manual_Value := #SPSel;
       #SPReal := #SPSel;
   END_IF;
END_REGION

REGION Network 26: **** 7.3 - Submodules - Machine **** Selection Manual Set-point
   // Selection Manual Set-point
   IF #ManualMode THEN #SPReal := #H_InOut.Manual_Value; END_IF;
END_REGION

NETWORK
TITLE = **** 7.3 - Submodules - Machine **** Reset Set-point in case of FaultA or B
// Reset Set-point in case of FaultA or B
      A(;
      A(;
      A     #AutoModeSel;
      A     #AlarmB;
      O;
      A     #AutoModeSel;
      A     #I_UpperLevelAlarmB;
      O     #AlarmA;
      O     #I_UpperLevelAlarmA;
      );
      JNB   _004;
      L     0.0;
      T     #SPReal;
      SET;
      SAVE;
      CLR;
_004: A     BR;
      );
      JNB   _005;
      L     0;
      T     #H_InOut.Manual_Value;
_005: NOP   0;

REGION Network 28: **** 7.3 - Submodule - Machine **** Frequency controller MRV (main reference value)
   // Frequency controller MRV (main reference value)
   // ENO of a box is taken as its EN; it also drops when the box reports an error
   #SPDINT := ROUND(#SPReal);
   #MRV_FC := #SPDINT;
END_REGION

REGION Network 29: **** 7.3 - Submodule - Machine **** Start Command Frequency controller
   // Start Command Frequency controller
   // Main reference value must be higher then 15 %
   #StartCmdFC := (#I_InterlockOk OR #ForcedMan) AND (#MRV_FC >= 15) AND #CmdRequest AND NOT #Contactor AND NOT #BypassForced;
END_REGION

REGION Network 30: **** 7.3 - Submodule - Machine **** Bypass Forced
   // Bypass Forced
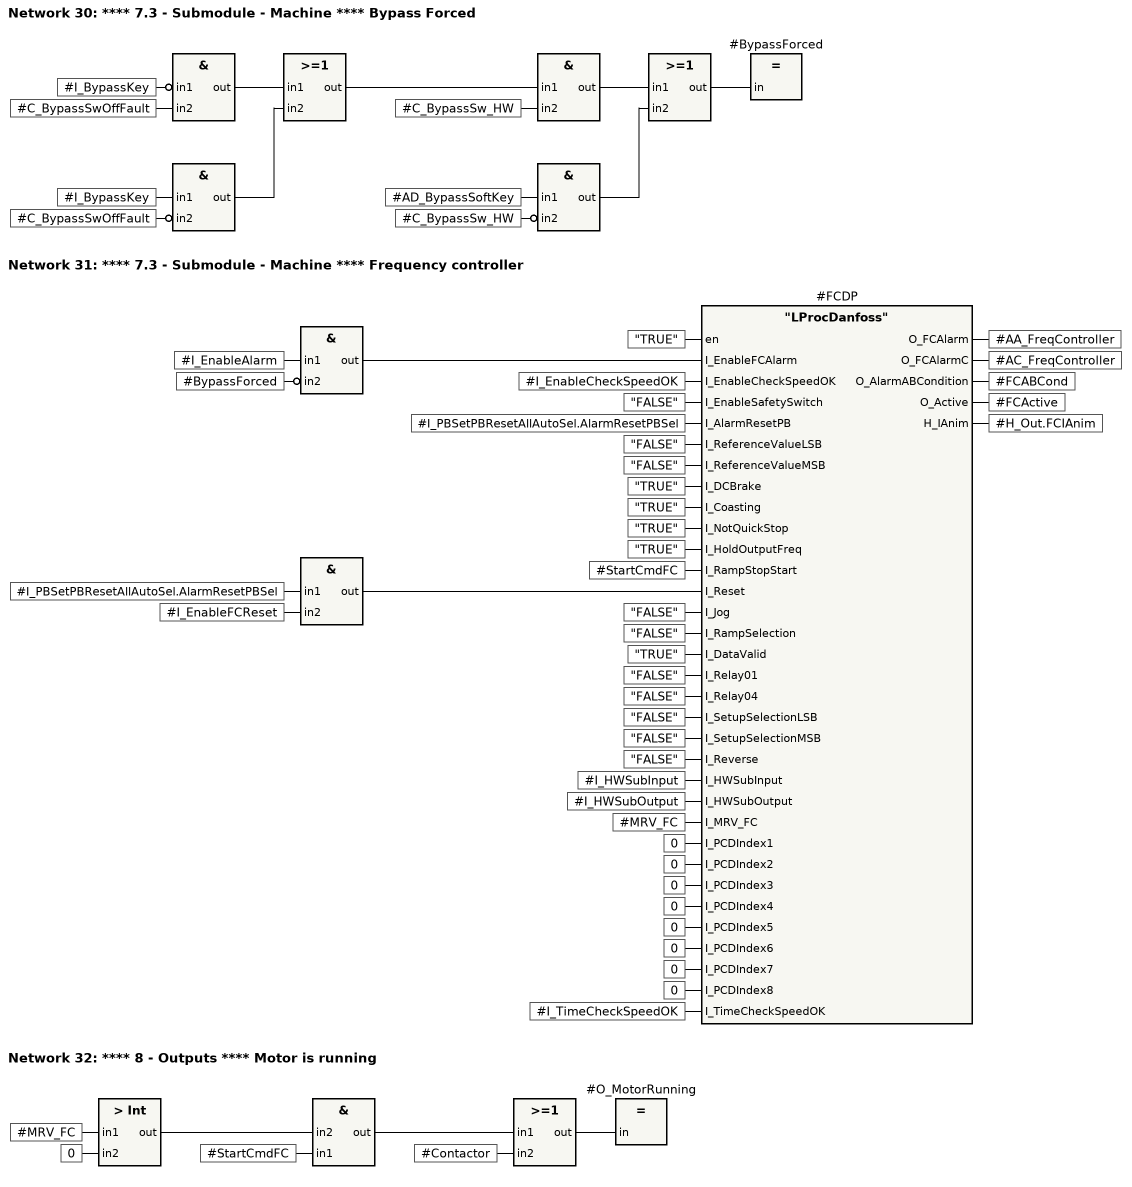
   #BypassForced := (((NOT #I_BypassKey AND #C_BypassSwOffFault) OR (#I_BypassKey AND NOT #C_BypassSwOffFault)) AND #C_BypassSw_HW) OR (#AD_BypassSoftKey AND NOT #C_BypassSw_HW);
END_REGION

REGION Network 31: **** 7.3 - Submodule - Machine **** Frequency controller
   // Frequency controller
   IF "TRUE" THEN
       #FCDP(I_EnableFCAlarm := #I_EnableAlarm AND NOT #BypassForced,   // "LProcDanfoss"
             I_EnableCheckSpeedOK := #I_EnableCheckSpeedOK,
             I_EnableSafetySwitch := "FALSE",
             I_AlarmResetPB := #I_PBSetPBResetAllAutoSel.AlarmResetPBSel,
             I_ReferenceValueLSB := "FALSE",
             I_ReferenceValueMSB := "FALSE",
             I_DCBrake := "TRUE",
             I_Coasting := "TRUE",
             I_NotQuickStop := "TRUE",
             I_HoldOutputFreq := "TRUE",
             I_RampStopStart := #StartCmdFC,
             I_Reset := #I_PBSetPBResetAllAutoSel.AlarmResetPBSel AND #I_EnableFCReset,
             I_Jog := "FALSE",
             I_RampSelection := "FALSE",
             I_DataValid := "TRUE",
             I_Relay01 := "FALSE",
             I_Relay04 := "FALSE",
             I_SetupSelectionLSB := "FALSE",
             I_SetupSelectionMSB := "FALSE",
             I_Reverse := "FALSE",
             I_HWSubInput := #I_HWSubInput,
             I_HWSubOutput := #I_HWSubOutput,
             I_MRV_FC := #MRV_FC,
             I_PCDIndex1 := 0,
             I_PCDIndex2 := 0,
             I_PCDIndex3 := 0,
             I_PCDIndex4 := 0,
             I_PCDIndex5 := 0,
             I_PCDIndex6 := 0,
             I_PCDIndex7 := 0,
             I_PCDIndex8 := 0,
             I_TimeCheckSpeedOK := #I_TimeCheckSpeedOK,
             O_FCAlarm => #AA_FreqController,
             O_FCAlarmC => #AC_FreqController,
             O_AlarmABCondition => #FCABCond,
             O_Active => #FCActive,
             H_IAnim => #H_Out.FCIAnim);
   END_IF;
END_REGION

REGION Network 32: **** 8 - Outputs **** Motor is running
   // Motor is running
   #O_MotorRunning := ((#MRV_FC > 0) AND #StartCmdFC) OR #Contactor;
END_REGION

REGION Network 33: **** 7.3 - Submodule - Machine **** Bypass Contactor
   // Bypass Contactor
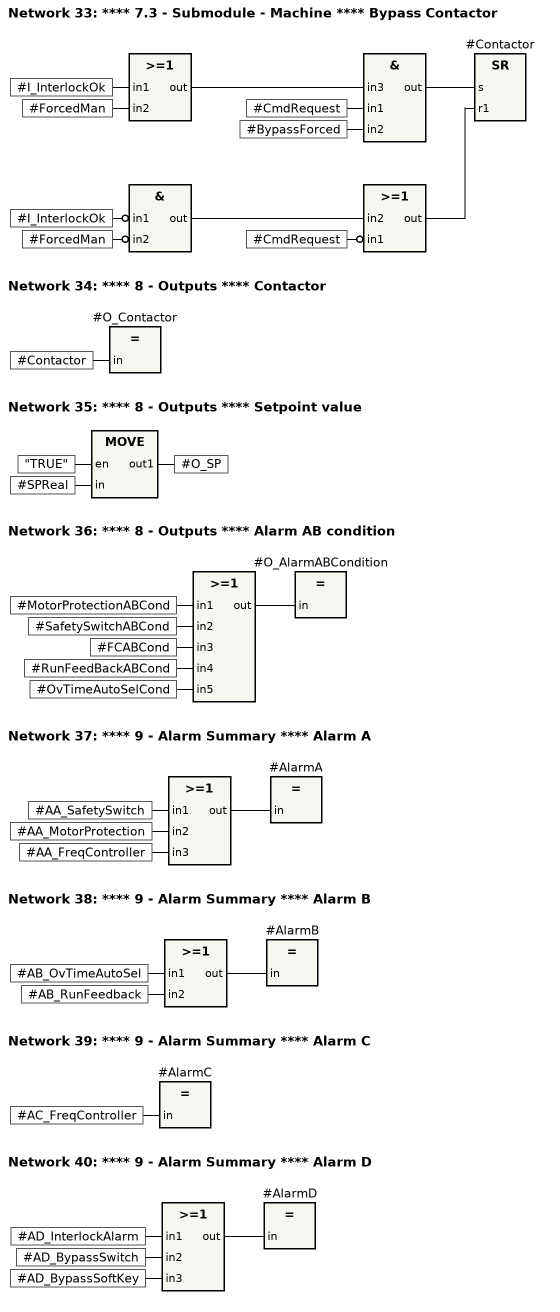
   IF (#I_InterlockOk OR #ForcedMan) AND #CmdRequest AND #BypassForced THEN
       #Contactor := TRUE;   // SR flip-flop
   END_IF;
   IF (NOT #I_InterlockOk AND NOT #ForcedMan) OR NOT #CmdRequest THEN #Contactor := FALSE; END_IF;
END_REGION

REGION Network 34: **** 8 - Outputs **** Contactor
   // Contactor
   #O_Contactor := #Contactor;
END_REGION

REGION Network 35: **** 8 - Outputs **** Setpoint value
   // Setpoint value
   IF "TRUE" THEN #O_SP := #SPReal; END_IF;
END_REGION

REGION Network 36: **** 8 - Outputs **** Alarm AB condition
   // Alarm AB Condition
   #O_AlarmABCondition := #MotorProtectionABCond OR #SafetySwitchABCond OR #FCABCond OR #RunFeedBackABCond OR #OvTimeAutoSelCond;
END_REGION

REGION Network 37: **** 9 - Alarm Summary **** Alarm A
   // Alarm A
   #AlarmA := #AA_SafetySwitch OR #AA_MotorProtection OR #AA_FreqController;
END_REGION

REGION Network 38: **** 9 - Alarm Summary **** Alarm B
   // Alarm B
   #AlarmB := #AB_OvTimeAutoSel OR #AB_RunFeedback;
END_REGION

REGION Network 39: **** 9 - Alarm Summary **** Alarm C
   // Alarm C
   #AlarmC := #AC_FreqController;
END_REGION

REGION Network 40: **** 9 - Alarm Summary **** Alarm D
   // Alarm D
   #AlarmD := #AD_InterlockAlarm OR #AD_BypassSwitch OR #AD_BypassSoftKey;
END_REGION

REGION Network 41: **** 9.1 - Alarm Output **** Alarm A
   // Alarm A
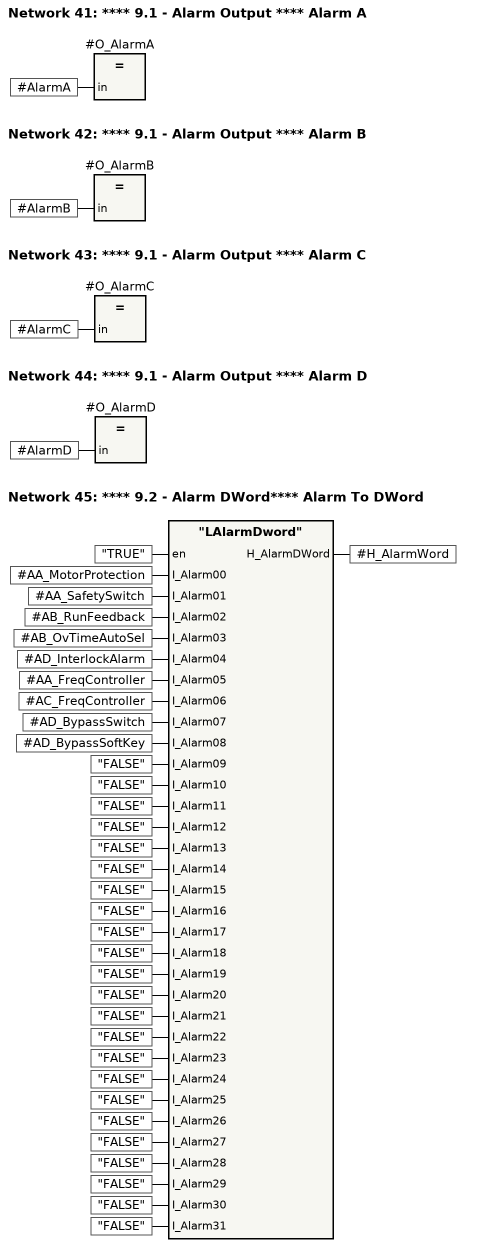
   #O_AlarmA := #AlarmA;
END_REGION

REGION Network 42: **** 9.1 - Alarm Output **** Alarm B
   // Alarm B
   #O_AlarmB := #AlarmB;
END_REGION

REGION Network 43: **** 9.1 - Alarm Output **** Alarm C
   // Alarm C
   #O_AlarmC := #AlarmC;
END_REGION

REGION Network 44: **** 9.1 - Alarm Output **** Alarm D
   // Alarm D
   #O_AlarmD := #AlarmD;
END_REGION

REGION Network 45: **** 9.2 - Alarm DWord**** Alarm To DWord
   // Alarm Word
   IF "TRUE" THEN
       "LAlarmDword"(I_Alarm00 := #AA_MotorProtection,
                     I_Alarm01 := #AA_SafetySwitch,
                     I_Alarm02 := #AB_RunFeedback,
                     I_Alarm03 := #AB_OvTimeAutoSel,
                     I_Alarm04 := #AD_InterlockAlarm,
                     I_Alarm05 := #AA_FreqController,
                     I_Alarm06 := #AC_FreqController,
                     I_Alarm07 := #AD_BypassSwitch,
                     I_Alarm08 := #AD_BypassSoftKey,
                     I_Alarm09 := "FALSE",
                     I_Alarm10 := "FALSE",
                     I_Alarm11 := "FALSE",
                     I_Alarm12 := "FALSE",
                     I_Alarm13 := "FALSE",
                     I_Alarm14 := "FALSE",
                     I_Alarm15 := "FALSE",
                     I_Alarm16 := "FALSE",
                     I_Alarm17 := "FALSE",
                     I_Alarm18 := "FALSE",
                     I_Alarm19 := "FALSE",
                     I_Alarm20 := "FALSE",
                     I_Alarm21 := "FALSE",
                     I_Alarm22 := "FALSE",
                     I_Alarm23 := "FALSE",
                     I_Alarm24 := "FALSE",
                     I_Alarm25 := "FALSE",
                     I_Alarm26 := "FALSE",
                     I_Alarm27 := "FALSE",
                     I_Alarm28 := "FALSE",
                     I_Alarm29 := "FALSE",
                     I_Alarm30 := "FALSE",
                     I_Alarm31 := "FALSE",
                     H_AlarmDWord => #H_AlarmWord);
   END_IF;
END_REGION
END_FUNCTION_BLOCK
